TYPE "ValveMachine_DataOut"
VERSION : 0.1
// Block: ValveMachine_DataOut
   STRUCT
      RestSolenoid : Bool;
      WorkSolenoid : Bool;
   END_STRUCT;

END_TYPE
